{attribute addProperty BoxType "CU1128--0000"}
{attribute addProperty Id "A_0005_CU1128_0000_0001A_0005_CU1128_0000_0001_D0E37FC3960120A_0004_CU1128_0000_0000_2_CU1128_BCU1128_179A0949162A_0004_CU1128_0000_0000_3_CU1128_CCU1128_179A0949162"}
{attribute addProperty CRC "662588022"}
{attribute addProperty SizeInBites "992"}
{attribute addProperty SizeInBytes "124"}
TYPE A_0004_CU1128_0000_0000_277E4A76 EXTENDS CU1128_179A0949 :
STRUCT
	{attribute addProperty Name "A_0005_CU1128_0000_0001"}
	A_0005_CU1128_0000_0001 : A_0005_CU1128_0000_0001_D0E37FC3;
	{attribute addProperty Name "A_0004_CU1128_0000_0000_2_CU1128_B"}
	A_0004_CU1128_0000_0000_2_CU1128_B : CU1128_179A0949;
	{attribute addProperty Name "A_0004_CU1128_0000_0000_3_CU1128_C"}
	A_0004_CU1128_0000_0000_3_CU1128_C : CU1128_179A0949;
END_STRUCT
END_TYPE

(* stored: Version 1.2.0.0, ProductVersion 3.1.4024.9
   DUT A_0004_CU1128_0000_0000_277E4A76: Id {96e253eb-a520-464f-ba9d-47585b914ca8} *)
